// TIA Portal V16 export
// export: Created 2021-11-12T13:52:02.1012746Z, ExportSetting WithDefaults, DisplayName Totally Integrated Automation Portal, DisplayVersion V16 Update 3, DisplayName TIA Portal Version Control Interface, DisplayVersion V16 Update 2, DisplayName TIA Portal Openness, DisplayVersion V16 Update 3, DisplayName SINAMICS Startdrive Advanced, DisplayVersion V16 Update 5, DisplayName SINAMICS Startdrive G130, G150, S120, S150, SINAMICS MV, S210, DisplayVersion V16 Update 5, DisplayName SINAMICS Startdrive G110M, G120, G120C, G120D, G120P, G115D, DisplayVersion V16 Update 5, DisplayName STEP 7 Professional, DisplayVersion V16 Update 3, DisplayName STEP 7 Safety, DisplayVersion V16, DisplayName WinCC UA Professional, DisplayVersion V16 Update 3
FUNCTION_BLOCK "STD_System"   // FB2, LAD
TITLE = STD_System
{ S7_Optimized_Access := 'TRUE' }
VERSION : 0.1
// MICE Wood template block
// Block for basic system function
// Set log.0, log.1
// Pulses and signals for blinking
// Commissioning signals
// ................................
// Version             Date                    Created by                    Comment
// 0.1                     31.1.2018           MSi                                 Initial version
// 0.2                     11.5.2018           MSi                                 Added pulse 500ms after PLC startup
// 1.0                     6.9. 2018            MSt                                Renamed from FB_System to STD_System
// stored: AutoNumber false, IsIECCheckEnabled false, IsRetainMemResEnabled false, MemoryReserve 100, SetENOAutomatically false, UDAEnableTagReadback false
   VAR
      SB1STDEdge_100ms : Bool;
      SB1STDEdge_200ms : Bool;
      SB1STDEdge_400ms : Bool;
      SB1STDEdge_500ms : Bool;
      SB1STDEdge_800ms : Bool;
      SB1STDEdge_1s : Bool;
      SB1STDEdge_1600ms : Bool;
      SB1STDEdge_2s : Bool;
      ST_TOFPulseEach10s { S7_SetPoint := 'True'} : TOF_TIME;
      ST_TOFPulseEach60s { S7_SetPoint := 'True'} : TOF_TIME;
      ST_TOFPulseEach600s { S7_SetPoint := 'True'} : TOF_TIME;
      ST_TOFPulseEach3600s { S7_SetPoint := 'True'} : TOF_TIME;
      ST_TONBlinking300ms { S7_SetPoint := 'True'} : TON_TIME;
      ST_TOFBlinking300ms { S7_SetPoint := 'True'} : TOF_TIME;
      ST_TONBlinking1sOn2sOff { S7_SetPoint := 'True'} : TON_TIME;
      ST_TOFBlinking1sOn2sOff { S7_SetPoint := 'True'} : TOF_TIME;
      ST_TOFDelayPulse500ms { S7_SetPoint := 'True'} : TOF_TIME;
   END_VAR
   VAR_TEMP   // added for the SCL form of the ladder/FBD networks
      _w1 : Bool;
      _w2 : Bool;
      _w3 : Bool;
      _w4 : Bool;
      _w5 : Bool;
      _w6 : Bool;
      _w7 : Bool;
      _w8 : Bool;
   END_VAR
BEGIN

REGION Network 1: Reset safety bypass Data block signals
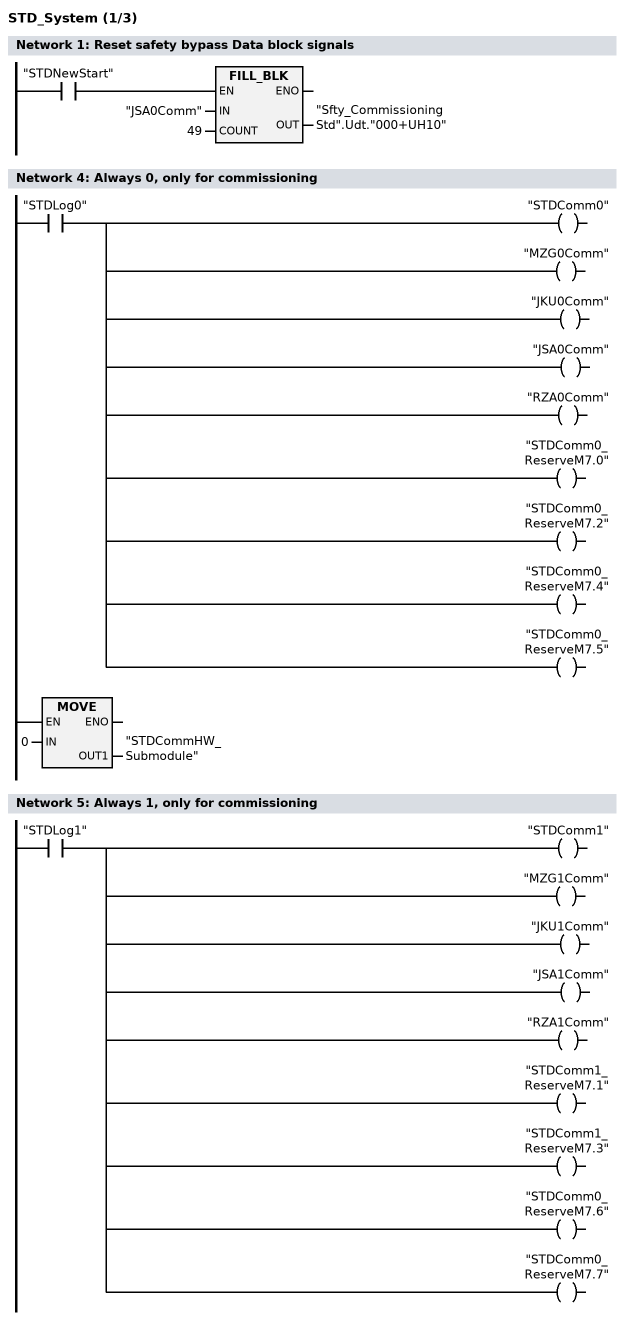
   RUNG wire#powerrail
      Contact( "STDNewStart" )
      FillBlockI(in := "JSA0Comm", count := 49, out => "Sfty_CommissioningStd".Udt."000+UH10")
   END_RUNG
   // the same network as SCL:
   IF "STDNewStart" THEN
       FILL_BLK(IN := "JSA0Comm", COUNT := 49, OUT => "Sfty_CommissioningStd".Udt."000+UH10");
   END_IF;
END_REGION

REGION Network 2: Always 0
   // Direct on CPU - HW config
END_REGION

REGION Network 3: Always 1
   // Direct on CPU - HW config
END_REGION

REGION Network 4: Always 0, only for commissioning
   RUNG wire#powerrail
      Contact( "STDLog0" )
      wire#w1
      Coil( "STDComm0" )
   END_RUNG
   RUNG wire#w1
      Coil( "MZG0Comm" )
   END_RUNG
   RUNG wire#w1
      Coil( "JKU0Comm" )
   END_RUNG
   RUNG wire#w1
      Coil( "JSA0Comm" )
   END_RUNG
   RUNG wire#w1
      Coil( "RZA0Comm" )
   END_RUNG
   RUNG wire#w1
      Coil( "STDComm0_ReserveM7.0" )
   END_RUNG
   RUNG wire#w1
      Coil( "STDComm0_ReserveM7.2" )
   END_RUNG
   RUNG wire#w1
      Coil( "STDComm0_ReserveM7.4" )
   END_RUNG
   RUNG wire#w1
      Coil( "STDComm0_ReserveM7.5" )
   END_RUNG
   RUNG wire#powerrail
      Move(in := 0, out1 => "STDCommHW_Submodule")
   END_RUNG
   // the same network as SCL:
   "STDComm0" := "STDLog0";
   "MZG0Comm" := "STDLog0";
   "JKU0Comm" := "STDLog0";
   "JSA0Comm" := "STDLog0";
   "RZA0Comm" := "STDLog0";
   "STDComm0_ReserveM7.0" := "STDLog0";
   "STDComm0_ReserveM7.2" := "STDLog0";
   "STDComm0_ReserveM7.4" := "STDLog0";
   "STDComm0_ReserveM7.5" := "STDLog0";
   "STDCommHW_Submodule" := 0;
END_REGION

REGION Network 5: Always 1, only for commissioning
   RUNG wire#powerrail
      Contact( "STDLog1" )
      wire#w1
      Coil( "STDComm1" )
   END_RUNG
   RUNG wire#w1
      Coil( "MZG1Comm" )
   END_RUNG
   RUNG wire#w1
      Coil( "JKU1Comm" )
   END_RUNG
   RUNG wire#w1
      Coil( "JSA1Comm" )
   END_RUNG
   RUNG wire#w1
      Coil( "RZA1Comm" )
   END_RUNG
   RUNG wire#w1
      Coil( "STDComm1_ReserveM7.1" )
   END_RUNG
   RUNG wire#w1
      Coil( "STDComm1_ReserveM7.3" )
   END_RUNG
   RUNG wire#w1
      Coil( "STDComm0_ReserveM7.6" )
   END_RUNG
   RUNG wire#w1
      Coil( "STDComm0_ReserveM7.7" )
   END_RUNG
   // the same network as SCL:
   "STDComm1" := "STDLog1";
   "MZG1Comm" := "STDLog1";
   "JKU1Comm" := "STDLog1";
   "JSA1Comm" := "STDLog1";
   "RZA1Comm" := "STDLog1";
   "STDComm1_ReserveM7.1" := "STDLog1";
   "STDComm1_ReserveM7.3" := "STDLog1";
   "STDComm0_ReserveM7.6" := "STDLog1";
   "STDComm0_ReserveM7.7" := "STDLog1";
END_REGION

REGION Network 6: PLC start up, 1 cycle active
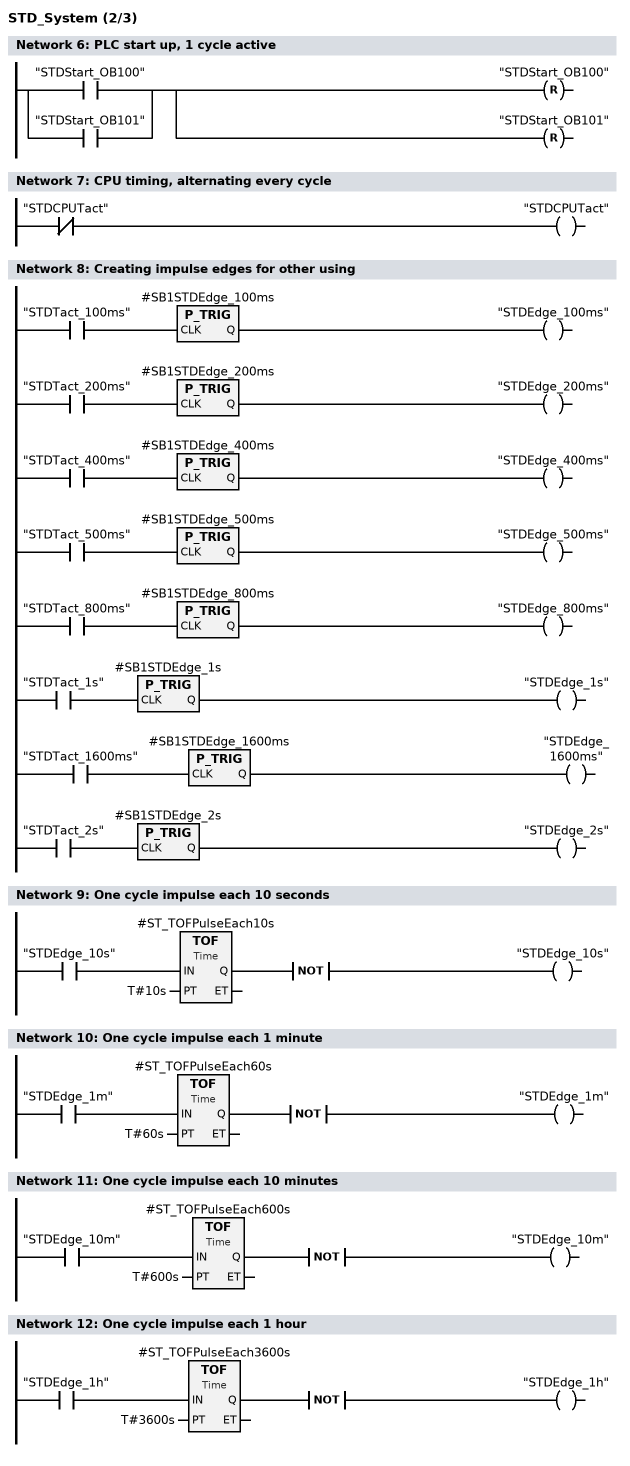
   RUNG wire#powerrail
      Contact( "STDStart_OB100" )
      wire#w1
      R_Coil( "STDStart_OB100" )
   END_RUNG
   RUNG wire#powerrail
      Contact( "STDStart_OB101" )
   END_RUNG wire#w1
   RUNG wire#w1
      R_Coil( "STDStart_OB101" )
   END_RUNG
   // the same network as SCL:
   #_w1 := "STDStart_OB100" OR "STDStart_OB101";
   IF #_w1 THEN
       "STDStart_OB100" := FALSE;
       "STDStart_OB101" := FALSE;
   END_IF;
END_REGION

REGION Network 7: CPU timing, alternating every cycle
   RUNG wire#powerrail
      I_Contact( "STDCPUTact" )
      Coil( "STDCPUTact" )
   END_RUNG
   // the same network as SCL:
   "STDCPUTact" := NOT "STDCPUTact";
END_REGION

REGION Network 8: Creating impulse edges for other using
   RUNG wire#powerrail
      Contact( "STDTact_100ms" )
      P_Trig( #SB1STDEdge_100ms )
      Coil( "STDEdge_100ms" )
   END_RUNG
   RUNG wire#powerrail
      Contact( "STDTact_200ms" )
      P_Trig( #SB1STDEdge_200ms )
      Coil( "STDEdge_200ms" )
   END_RUNG
   RUNG wire#powerrail
      Contact( "STDTact_400ms" )
      P_Trig( #SB1STDEdge_400ms )
      Coil( "STDEdge_400ms" )
   END_RUNG
   RUNG wire#powerrail
      Contact( "STDTact_500ms" )
      P_Trig( #SB1STDEdge_500ms )
      Coil( "STDEdge_500ms" )
   END_RUNG
   RUNG wire#powerrail
      Contact( "STDTact_800ms" )
      P_Trig( #SB1STDEdge_800ms )
      Coil( "STDEdge_800ms" )
   END_RUNG
   RUNG wire#powerrail
      Contact( "STDTact_1s" )
      P_Trig( #SB1STDEdge_1s )
      Coil( "STDEdge_1s" )
   END_RUNG
   RUNG wire#powerrail
      Contact( "STDTact_1600ms" )
      P_Trig( #SB1STDEdge_1600ms )
      Coil( "STDEdge_1600ms" )
   END_RUNG
   RUNG wire#powerrail
      Contact( "STDTact_2s" )
      P_Trig( #SB1STDEdge_2s )
      Coil( "STDEdge_2s" )
   END_RUNG
   // the same network as SCL:
   #_w1 := "STDTact_100ms" AND NOT #SB1STDEdge_100ms;   // rising edge
   #SB1STDEdge_100ms := "STDTact_100ms";
   "STDEdge_100ms" := #_w1;
   #_w2 := "STDTact_200ms" AND NOT #SB1STDEdge_200ms;   // rising edge
   #SB1STDEdge_200ms := "STDTact_200ms";
   "STDEdge_200ms" := #_w2;
   #_w3 := "STDTact_400ms" AND NOT #SB1STDEdge_400ms;   // rising edge
   #SB1STDEdge_400ms := "STDTact_400ms";
   "STDEdge_400ms" := #_w3;
   #_w4 := "STDTact_500ms" AND NOT #SB1STDEdge_500ms;   // rising edge
   #SB1STDEdge_500ms := "STDTact_500ms";
   "STDEdge_500ms" := #_w4;
   #_w5 := "STDTact_800ms" AND NOT #SB1STDEdge_800ms;   // rising edge
   #SB1STDEdge_800ms := "STDTact_800ms";
   "STDEdge_800ms" := #_w5;
   #_w6 := "STDTact_1s" AND NOT #SB1STDEdge_1s;   // rising edge
   #SB1STDEdge_1s := "STDTact_1s";
   "STDEdge_1s" := #_w6;
   #_w7 := "STDTact_1600ms" AND NOT #SB1STDEdge_1600ms;   // rising edge
   #SB1STDEdge_1600ms := "STDTact_1600ms";
   "STDEdge_1600ms" := #_w7;
   #_w8 := "STDTact_2s" AND NOT #SB1STDEdge_2s;   // rising edge
   #SB1STDEdge_2s := "STDTact_2s";
   "STDEdge_2s" := #_w8;
END_REGION

REGION Network 9: One cycle impulse each 10 seconds
   RUNG wire#powerrail
      Contact( "STDEdge_10s" )
      { S7_Templates := "time_type := Time" } #ST_TOFPulseEach10s.TOF(pt := T#10s, et =>)
      Not()
      Coil( "STDEdge_10s" )
   END_RUNG
   // the same network as SCL:
   #ST_TOFPulseEach10s(IN := "STDEdge_10s", PT := T#10s);   // TOF
   "STDEdge_10s" := NOT #ST_TOFPulseEach10s.Q;
END_REGION

REGION Network 10: One cycle impulse each 1 minute
   RUNG wire#powerrail
      Contact( "STDEdge_1m" )
      { S7_Templates := "time_type := Time" } #ST_TOFPulseEach60s.TOF(pt := T#60s, et =>)
      Not()
      Coil( "STDEdge_1m" )
   END_RUNG
   // the same network as SCL:
   #ST_TOFPulseEach60s(IN := "STDEdge_1m", PT := T#60s);   // TOF
   "STDEdge_1m" := NOT #ST_TOFPulseEach60s.Q;
END_REGION

REGION Network 11: One cycle impulse each 10 minutes
   RUNG wire#powerrail
      Contact( "STDEdge_10m" )
      { S7_Templates := "time_type := Time" } #ST_TOFPulseEach600s.TOF(pt := T#600s, et =>)
      Not()
      Coil( "STDEdge_10m" )
   END_RUNG
   // the same network as SCL:
   #ST_TOFPulseEach600s(IN := "STDEdge_10m", PT := T#600s);   // TOF
   "STDEdge_10m" := NOT #ST_TOFPulseEach600s.Q;
END_REGION

REGION Network 12: One cycle impulse each 1 hour
   RUNG wire#powerrail
      Contact( "STDEdge_1h" )
      { S7_Templates := "time_type := Time" } #ST_TOFPulseEach3600s.TOF(pt := T#3600s, et =>)
      Not()
      Coil( "STDEdge_1h" )
   END_RUNG
   // the same network as SCL:
   #ST_TOFPulseEach3600s(IN := "STDEdge_1h", PT := T#3600s);   // TOF
   "STDEdge_1h" := NOT #ST_TOFPulseEach3600s.Q;
END_REGION

REGION Network 13: Blinking 0,3s ON / 0,3s OFF - active alarm
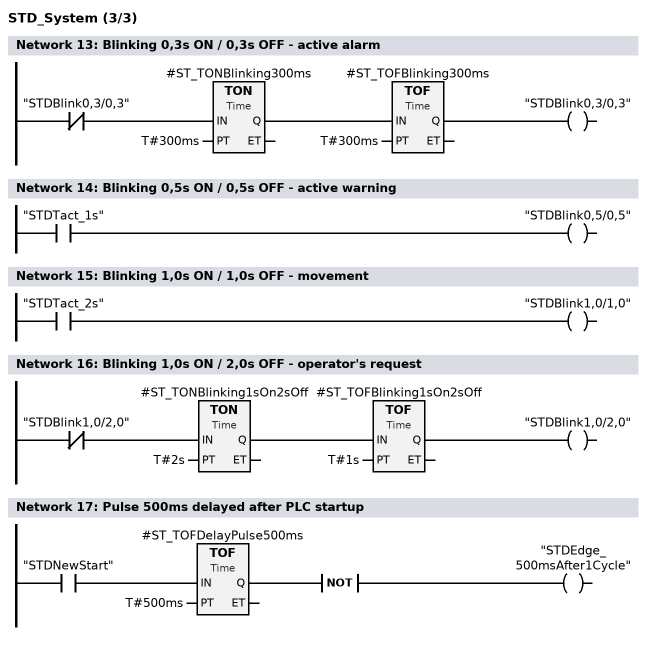
   RUNG wire#powerrail
      I_Contact( "STDBlink0,3/0,3" )
      { S7_Templates := "time_type := Time" } #ST_TONBlinking300ms.TON(pt := T#300ms, et =>)
      { S7_Templates := "time_type := Time" } #ST_TOFBlinking300ms.TOF(pt := T#300ms, et =>)
      Coil( "STDBlink0,3/0,3" )
   END_RUNG
   // the same network as SCL:
   #ST_TONBlinking300ms(IN := NOT "STDBlink0,3/0,3", PT := T#300ms);   // TON
   #ST_TOFBlinking300ms(IN := #ST_TONBlinking300ms.Q, PT := T#300ms);   // TOF
   "STDBlink0,3/0,3" := #ST_TOFBlinking300ms.Q;
END_REGION

REGION Network 14: Blinking 0,5s ON / 0,5s OFF - active warning
   RUNG wire#powerrail
      Contact( "STDTact_1s" )
      Coil( "STDBlink0,5/0,5" )
   END_RUNG
   // the same network as SCL:
   "STDBlink0,5/0,5" := "STDTact_1s";
END_REGION

REGION Network 15: Blinking 1,0s ON / 1,0s OFF - movement
   RUNG wire#powerrail
      Contact( "STDTact_2s" )
      Coil( "STDBlink1,0/1,0" )
   END_RUNG
   // the same network as SCL:
   "STDBlink1,0/1,0" := "STDTact_2s";
END_REGION

REGION Network 16: Blinking 1,0s ON / 2,0s OFF - operator's request
   RUNG wire#powerrail
      I_Contact( "STDBlink1,0/2,0" )
      { S7_Templates := "time_type := Time" } #ST_TONBlinking1sOn2sOff.TON(pt := T#2s, et =>)
      { S7_Templates := "time_type := Time" } #ST_TOFBlinking1sOn2sOff.TOF(pt := T#1s, et =>)
      Coil( "STDBlink1,0/2,0" )
   END_RUNG
   // the same network as SCL:
   #ST_TONBlinking1sOn2sOff(IN := NOT "STDBlink1,0/2,0", PT := T#2s);   // TON
   #ST_TOFBlinking1sOn2sOff(IN := #ST_TONBlinking1sOn2sOff.Q, PT := T#1s);   // TOF
   "STDBlink1,0/2,0" := #ST_TOFBlinking1sOn2sOff.Q;
END_REGION

REGION Network 17: Pulse 500ms delayed after PLC startup
   RUNG wire#powerrail
      Contact( "STDNewStart" )
      { S7_Templates := "time_type := Time" } #ST_TOFDelayPulse500ms.TOF(pt := T#500ms, et =>)
      Not()
      Coil( "STDEdge_500msAfter1Cycle" )
   END_RUNG
   // the same network as SCL:
   #ST_TOFDelayPulse500ms(IN := "STDNewStart", PT := T#500ms);   // TOF
   "STDEdge_500msAfter1Cycle" := NOT #ST_TOFDelayPulse500ms.Q;
END_REGION
END_FUNCTION_BLOCK
